// Mitsubishi GX Works2 project: Group11   PLC: FX3G

// global labels: Global1
VAR_GLOBAL
  Start_Day AT X007 : BOOL;
  Start_Light AT Y000 : BOOL;
  Emergency AT X005 : BOOL;
  Storage_Light AT M4 : BOOL;
END_VAR
VAR_GLOBAL CONSTANT
  Oat_Min : INT := 400;
END_VAR
VAR_GLOBAL
  Oat_Storage AT D1100 : REAL;
  Oat_Storage_Light AT M1 : BOOL;
END_VAR
VAR_GLOBAL CONSTANT
  Pro_Min : INT := 320;
END_VAR
VAR_GLOBAL
  Pro_Storage AT D1200 : REAL;
  Pro_Storage_Light AT M2 : BOOL;
END_VAR
VAR_GLOBAL CONSTANT
  Honey_Min : INT := 160;
END_VAR
VAR_GLOBAL
  Honey_Storage AT D1300 : REAL;
  Hoeny_Storage_Light AT M3 : BOOL;
  Start_Blend AT X003 : BOOL;
  Analog_Input1 AT D8280 : INT;
  Analog_Light AT M7 : BOOL;
  Snack_Type AT D8000 : INT;
  Blend_Time AT TC5 : BOOL;
END_VAR
VAR_GLOBAL CONSTANT
  B_5Sec_Timer : INT := 50;
  Classic0_5 : INT := 6;
END_VAR
VAR_GLOBAL
  Classic_Snack_Light AT M8 : BOOL;
END_VAR
VAR_GLOBAL CONSTANT
  Pro6_10 : INT := 6;
END_VAR
VAR_GLOBAL
  Pro_Snack_Light AT M9 : BOOL;
  Blend_Time_TS AT TS5 : BOOL;
  Blend_Light AT Y003 : BOOL;
END_VAR
VAR_GLOBAL CONSTANT
  C_400 : INT := 6;
  CON_400 : INT := 400;
  CON_160 : INT := 160;
  CON_120 : INT := 120;
  CON_240 : INT := 240;
  CON_320 : INT := 320;
  Oat_User : INT := 1000;
END_VAR
VAR_GLOBAL
  Start_Cook AT X002 : BOOL;
  Cook_Light1 AT Y001 : BOOL;
  Cook_Light2 AT Y002 : BOOL;
  Cook_Time_Classic AT TC6 : BOOL;
END_VAR
VAR_GLOBAL CONSTANT
  C_4Sec_Timer_Classic : INT := 40;
END_VAR
VAR_GLOBAL
  Cook_Time_Classic_TS AT TS6 : BOOL;
  Cook_Time_Classic2 AT TC7 : BOOL;
  Cook_Time_Classic2_TS AT TS7 : BOOL;
  Cook_Time_Pro AT TC8 : BOOL;
END_VAR
VAR_GLOBAL CONSTANT
  C_5Sec_Timer_Pro : INT := 50;
END_VAR
VAR_GLOBAL
  Cook_Time_Pro_TS AT TS8 : BOOL;
  Cook_Time_Pro2 AT TC9 : BOOL;
  Cook_Time_Pro2_TS AT TS9 : BOOL;
  Flicker_Light_Classic AT M10 : BOOL;
  Flicker_Light_Pro AT M11 : BOOL;
  Flicker_Time1 AT TC1 : BOOL;
END_VAR
VAR_GLOBAL CONSTANT
  C_1Sec_Timer : INT := 10;
END_VAR
VAR_GLOBAL
  Cook_Time_TS1 AT TS1 : BOOL;
  Flicker_Light AT M10 : BOOL;
  Flicker_Time2 AT TC2 : BOOL;
  Cook_Time_TS2 AT TS2 : BOOL;
  Start_Pack AT X006 : BOOL;
  Pack_Snack AT X000 : BOOL;
  Pack_Snack_Light AT Y004 : BOOL;
  Counter_Pack AT CC1 : BOOL;
END_VAR
VAR_GLOBAL CONSTANT
  CON_8 : INT := 8;
END_VAR
VAR_GLOBAL
  CS_Pack AT CS1 : BOOL;
  Packeges_Num AT D1400 : REAL;
END_VAR
VAR_GLOBAL CONSTANT
  CON_1 : INT := 1;
  CON_10 : INT := 10;
END_VAR
VAR_GLOBAL
  Analog_Output AT D8282 : INT;
  Packeges_Num_Output AT D8100 : INT;
  Bigger6_Light AT M11 : BOOL;
  Not120_Light AT M12 : BOOL;
END_VAR
VAR_GLOBAL CONSTANT
  CON_40 : INT := 40;
END_VAR

// task Task_01 (event TRUE, interval 0, priority 31): POU_01

PROGRAM POU_01
(* structured ladder/FBD written out as ST: instructions are called as NAME(EN, inputs, outputs); _pN, _eN, _tN stand for wires *)
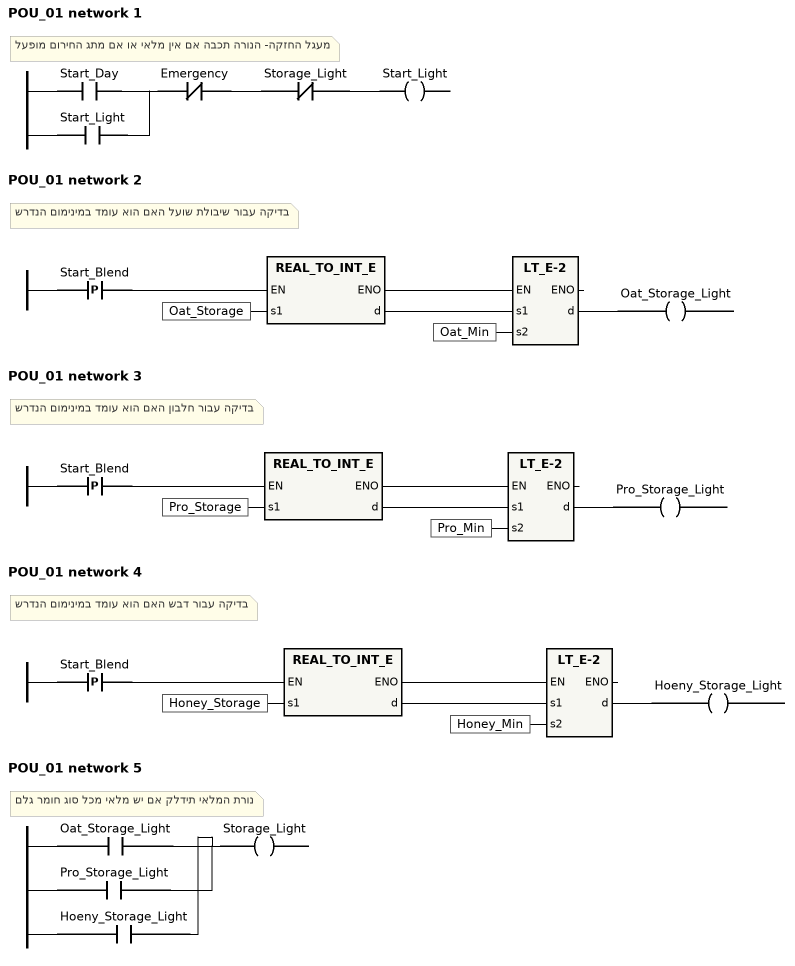
(* network 1 *)
(* מעגל החזקה- הנורה תכבה אם אין מלאי או אם מתג החירום מופעל *)
Start_Light := ((Start_Day OR Start_Light) AND NOT Emergency) AND NOT Storage_Light;
(* network 2 *)
(* בדיקה עבור שיבולת שועל האם הוא עומד במינימום הנדרש *)
_e2 := REAL_TO_INT_E(LDP(TRUE, Start_Blend), Oat_Storage, _t1);
LT_E(_e2, _t1, Oat_Min, _t3);
Oat_Storage_Light := _t3;
(* network 3 *)
(* בדיקה עבור חלבון האם הוא עומד במינימום הנדרש *)
_e2 := REAL_TO_INT_E(LDP(TRUE, Start_Blend), Pro_Storage, _t1);
LT_E(_e2, _t1, Pro_Min, _t3);
Pro_Storage_Light := _t3;
(* network 4 *)
(* בדיקה עבור דבש האם הוא עומד במינימום הנדרש *)
_e2 := REAL_TO_INT_E(LDP(TRUE, Start_Blend), Honey_Storage, _t1);
LT_E(_e2, _t1, Honey_Min, _t3);
Hoeny_Storage_Light := _t3;
(* network 5 *)
(* נורת המלאי תידלק אם יש מלאי מכל סוג חומר גלם *)
Storage_Light := Oat_Storage_Light OR Pro_Storage_Light OR Hoeny_Storage_Light;
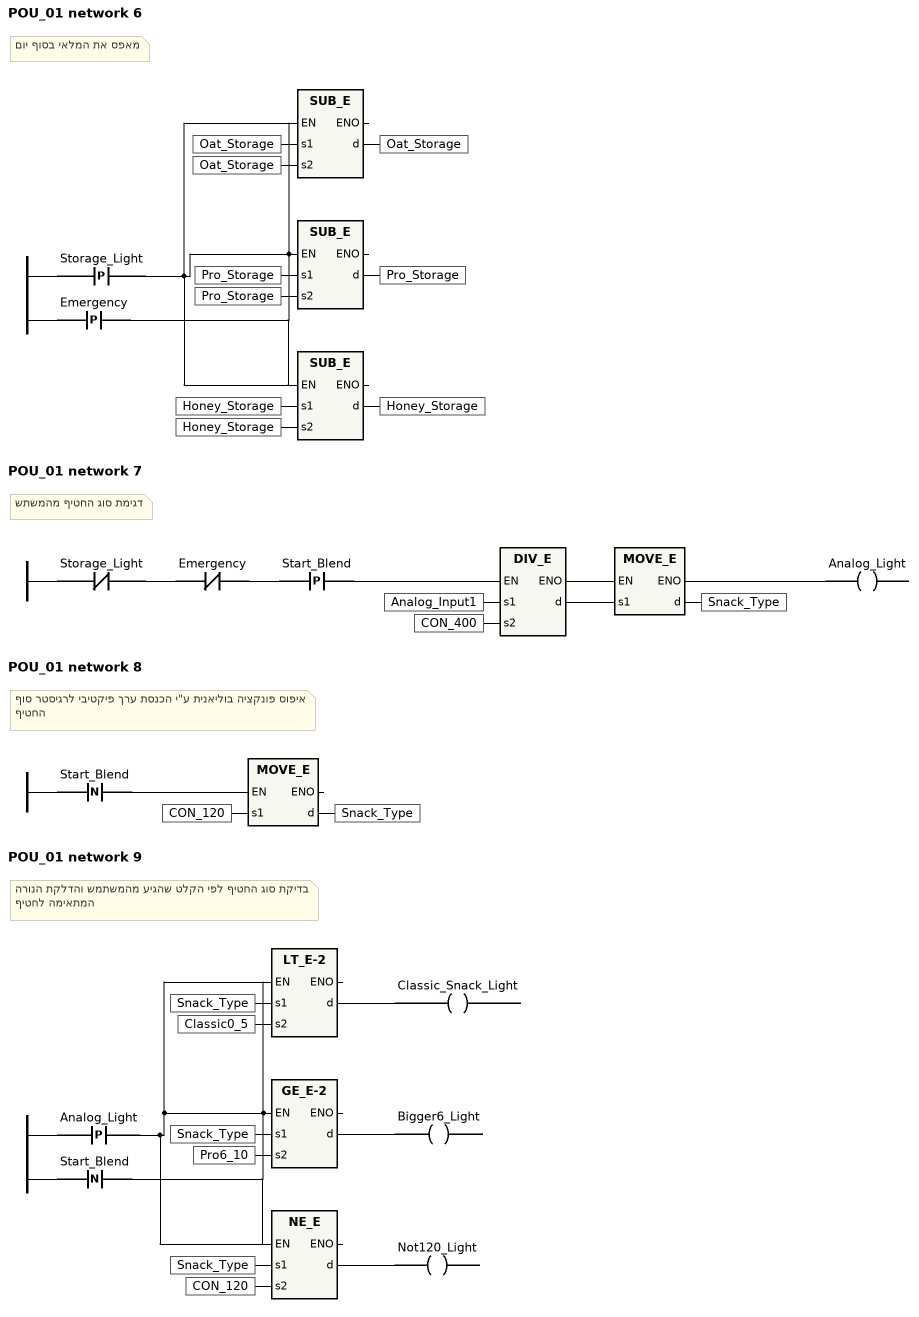
(* network 6 *)
(* מאפס את המלאי בסוף יום *)
_p1 := LDP(TRUE, Storage_Light) OR LDP(TRUE, Emergency);
SUB_E(_p1, Oat_Storage, Oat_Storage, Oat_Storage);
SUB_E(_p1, Pro_Storage, Pro_Storage, Pro_Storage);
SUB_E(_p1, Honey_Storage, Honey_Storage, Honey_Storage);
(* network 7 *)
(* דגימת סוג החטיף מהמשתש *)
_e2 := DIV_E(NOT Storage_Light AND NOT Emergency AND LDP(TRUE, Start_Blend), Analog_Input1, CON_400, _t1);
_e3 := MOVE_E(_e2, _t1, Snack_Type);
Analog_Light := _e3;
(* network 8 *)
(* איפוס פונקציה בוליאנית ע"י הכנסת ערך פיקטיבי לרגיסטר סוף החטיף *)
MOVE_E(LDF(TRUE, Start_Blend), CON_120, Snack_Type);
(* network 9 *)
(* בדיקת סוג החטיף לפי הקלט שהגיע מהמשתמש והדלקת הנורה המתאימה לחטיף *)
_p1 := LDP(TRUE, Analog_Light) OR LDF(TRUE, Start_Blend);
LT_E(_p1, Snack_Type, Classic0_5, _t2);
Classic_Snack_Light := _t2;
GE_E(_p1, Snack_Type, Pro6_10, _t3);
Bigger6_Light := _t3;
NE_E(_p1, Snack_Type, CON_120, _t4);
Not120_Light := _t4;
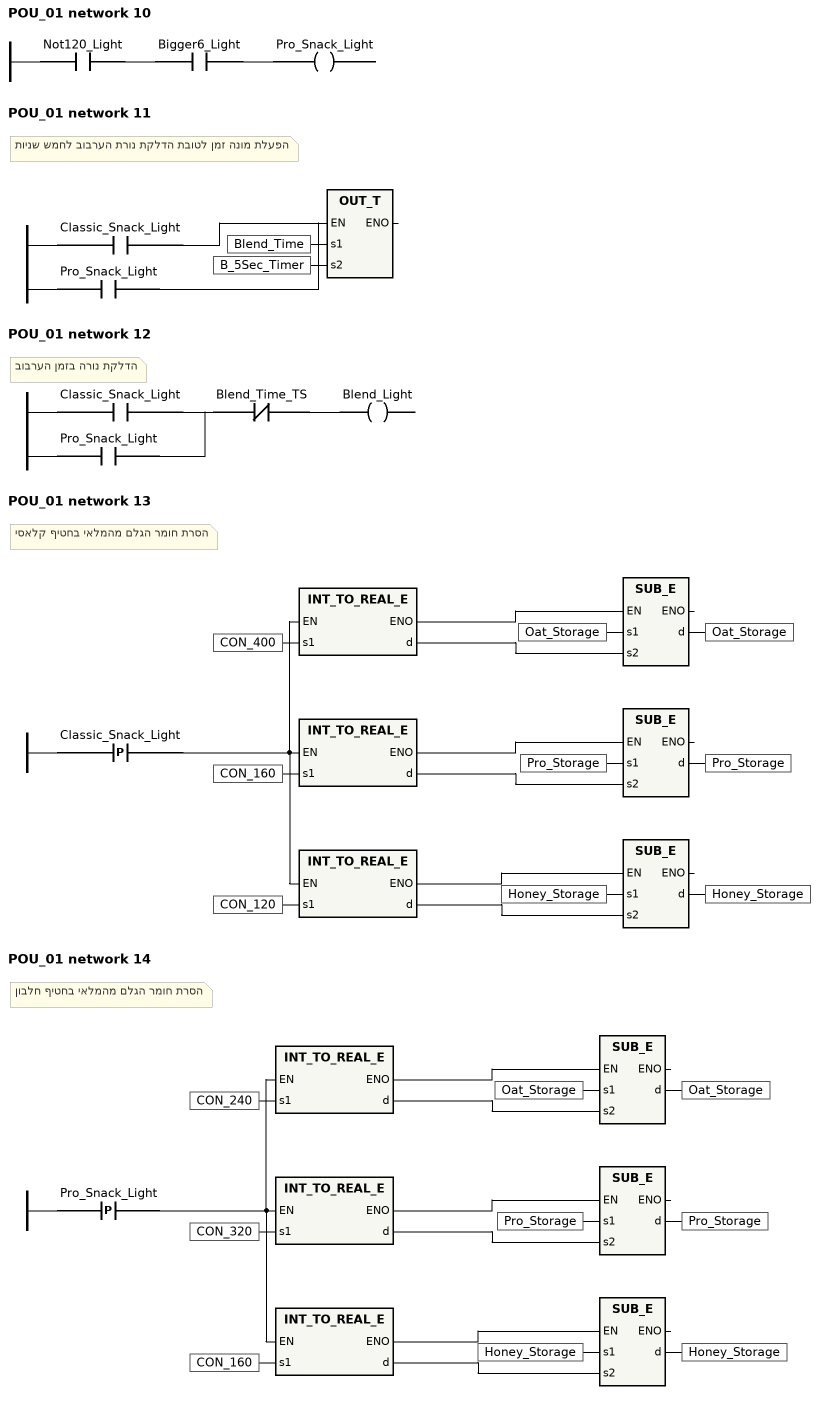
(* network 10 *)
Pro_Snack_Light := Not120_Light AND Bigger6_Light;
(* network 11 *)
(* הפעלת מונה זמן לטובת הדלקת נורת הערבוב לחמש שניות *)
OUT_T(Classic_Snack_Light OR Pro_Snack_Light, Blend_Time, B_5Sec_Timer);
(* network 12 *)
(* הדלקת נורה בזמן הערבוב *)
Blend_Light := (Classic_Snack_Light OR Pro_Snack_Light) AND NOT Blend_Time_TS;
(* network 13 *)
(* הסרת חומר הגלם מהמלאי בחטיף קלאסי *)
_p1 := LDP(TRUE, Classic_Snack_Light);
_e3 := INT_TO_REAL_E(_p1, CON_400, _t2);
SUB_E(_e3, Oat_Storage, _t2, Oat_Storage);
_e5 := INT_TO_REAL_E(_p1, CON_160, _t4);
SUB_E(_e5, Pro_Storage, _t4, Pro_Storage);
_e7 := INT_TO_REAL_E(_p1, CON_120, _t6);
SUB_E(_e7, Honey_Storage, _t6, Honey_Storage);
(* network 14 *)
(* הסרת חומר הגלם מהמלאי בחטיף חלבון *)
_p1 := LDP(TRUE, Pro_Snack_Light);
_e3 := INT_TO_REAL_E(_p1, CON_240, _t2);
SUB_E(_e3, Oat_Storage, _t2, Oat_Storage);
_e5 := INT_TO_REAL_E(_p1, CON_320, _t4);
SUB_E(_e5, Pro_Storage, _t4, Pro_Storage);
_e7 := INT_TO_REAL_E(_p1, CON_160, _t6);
SUB_E(_e7, Honey_Storage, _t6, Honey_Storage);
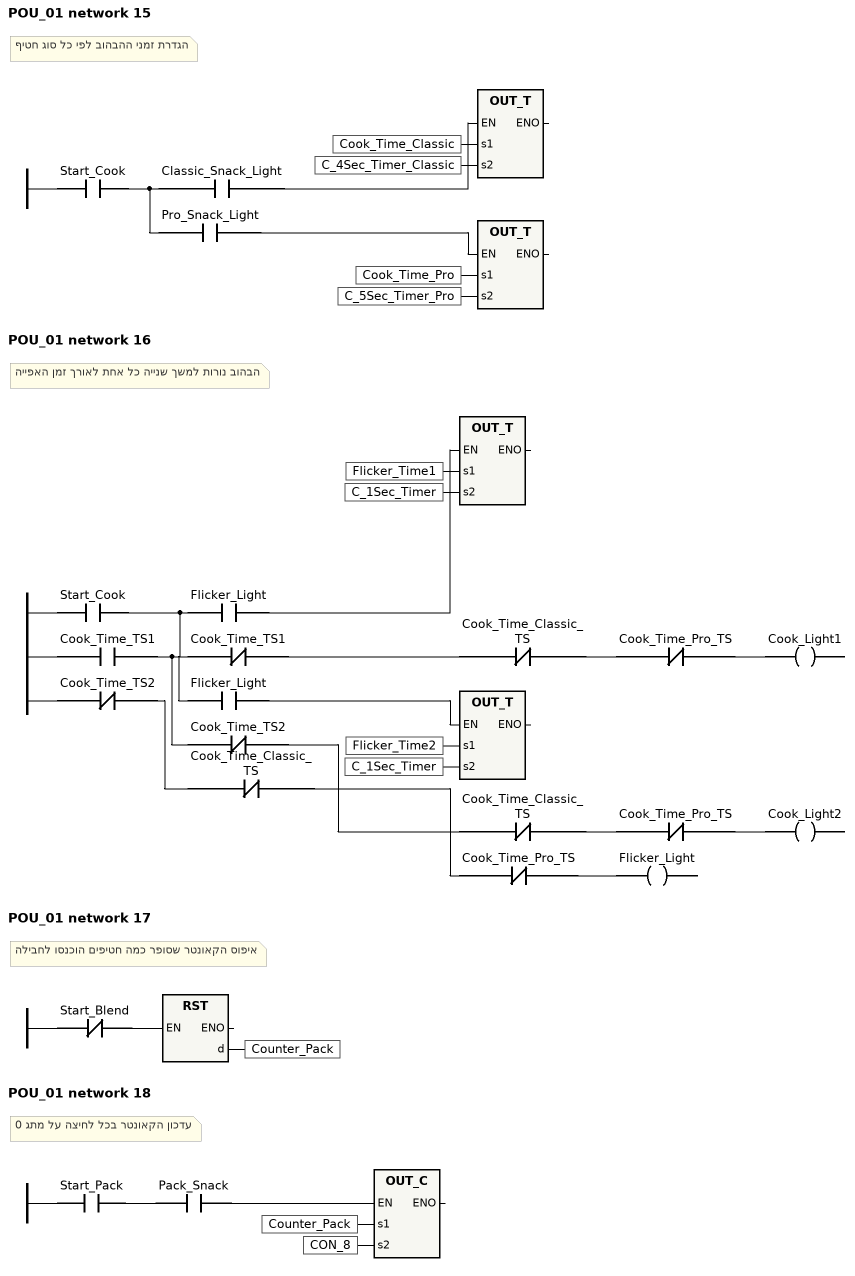
(* network 15 *)
(* הגדרת זמני ההבהוב לפי כל סוג חטיף *)
OUT_T(Start_Cook AND Classic_Snack_Light, Cook_Time_Classic, C_4Sec_Timer_Classic);
OUT_T(Start_Cook AND Pro_Snack_Light, Cook_Time_Pro, C_5Sec_Timer_Pro);
(* network 16 *)
(* הבהוב נורות למשך שנייה כל אחת לאורך זמן האפייה *)
OUT_T(Start_Cook AND Flicker_Light, Flicker_Time1, C_1Sec_Timer);
Cook_Light1 := Start_Cook AND NOT Cook_Time_TS1 AND NOT Cook_Time_Classic_TS AND NOT Cook_Time_Pro_TS;
OUT_T(Cook_Time_TS1 AND Flicker_Light, Flicker_Time2, C_1Sec_Timer);
Cook_Light2 := Cook_Time_TS1 AND NOT Cook_Time_TS2 AND NOT Cook_Time_Classic_TS AND NOT Cook_Time_Pro_TS;
Flicker_Light := NOT Cook_Time_TS2 AND NOT Cook_Time_Classic_TS AND NOT Cook_Time_Pro_TS;
(* network 17 *)
(* איפוס הקאונטר שסופר כמה חטיפים הוכנסו לחבילה *)
RST(NOT Start_Blend, Counter_Pack);
(* network 18 *)
(* עדכון הקאונטר בכל לחיצה על מתג 0 *)
OUT_C(Start_Pack AND Pack_Snack, Counter_Pack, CON_8);
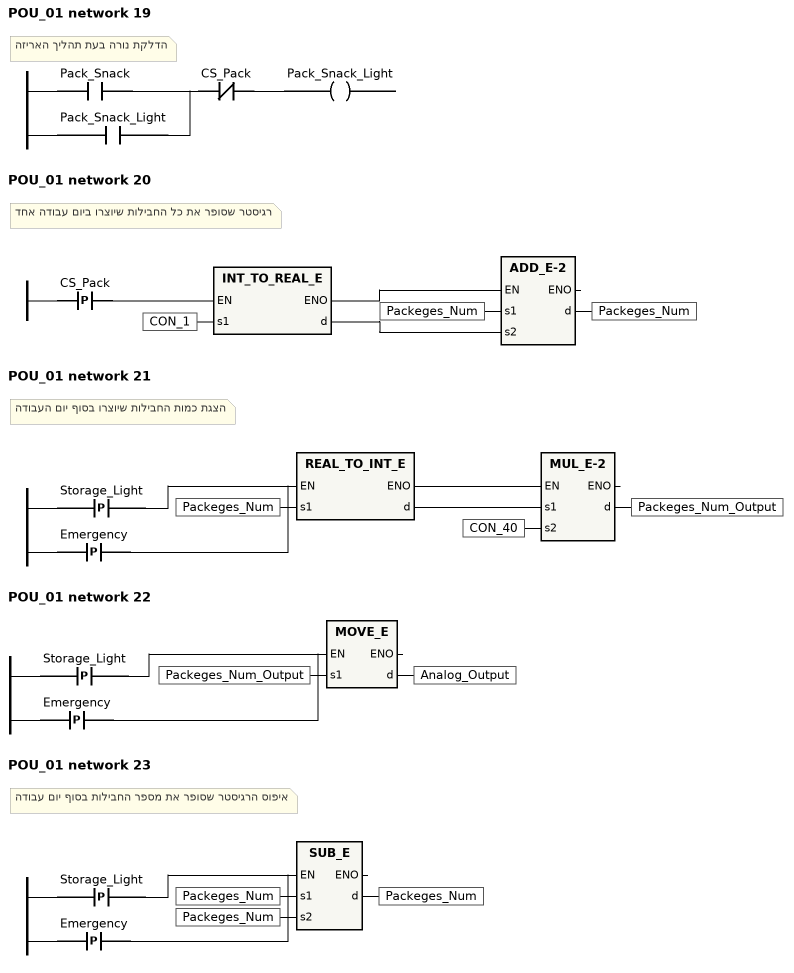
(* network 19 *)
(* הדלקת נורה בעת תהליך האריזה *)
Pack_Snack_Light := (Pack_Snack OR Pack_Snack_Light) AND NOT CS_Pack;
(* network 20 *)
(* רגיסטר שסופר את כל החבילות שיוצרו ביום עבודה אחד *)
_e2 := INT_TO_REAL_E(LDP(TRUE, CS_Pack), CON_1, _t1);
ADD_E(_e2, Packeges_Num, _t1, Packeges_Num);
(* network 21 *)
(* הצגת כמות החבילות שיוצרו בסוף יום העבודה *)
_e2 := REAL_TO_INT_E(LDP(TRUE, Storage_Light) OR LDP(TRUE, Emergency), Packeges_Num, _t1);
MUL_E(_e2, _t1, CON_40, Packeges_Num_Output);
(* network 22 *)
MOVE_E(LDP(TRUE, Storage_Light) OR LDP(TRUE, Emergency), Packeges_Num_Output, Analog_Output);
(* network 23 *)
(* איפוס הרגיסטר שסופר את מספר החבילות בסוף יום עבודה *)
SUB_E(LDP(TRUE, Storage_Light) OR LDP(TRUE, Emergency), Packeges_Num, Packeges_Num, Packeges_Num);
END_PROGRAM
